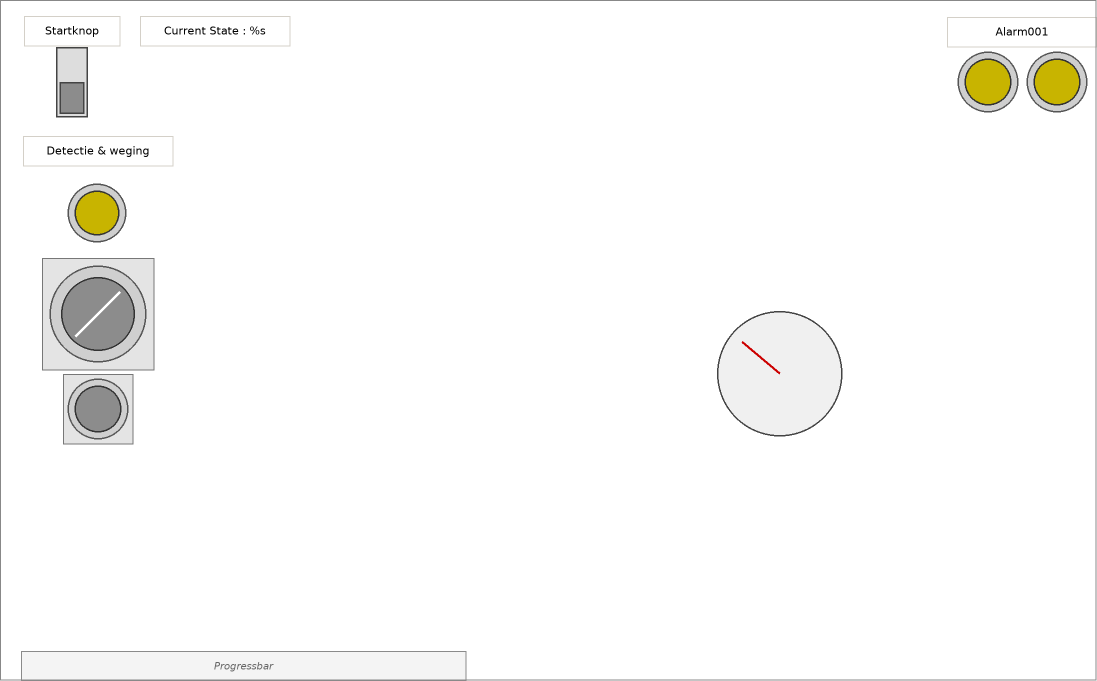
VISUALIZATION Overview  // 1097x681
    Meter180 (657,311 245x125), value: GVL.geschrevenSnelheid, style: Meter-Meter180-Gray, scale format: %.1f, scale 0..200
    Progressbar (21,651 445x30)
    Potentiometer360 (42,254 112x120), variable: GVL.weegcelWaarde, style: Potentiometer-Potentiometer360-Gray, scale format: %.1f, scale 0..100
        p2431819421: Outside
    PushSwitchLed (63,374 70x70), variable: GVL.LS_001, behaviour: TOGGLE, style: Switch-PushSwitchLed-Gray
    Lamp1 (63,178 68x70), variable: GVL.objectDetected, style: Lamp-Lamp1-Yellow
    Textfield (23,136 150x30), "Detectie & weging"
    Group (24,16 96x101)
        Textfield (0,0 96x30), "Startknop", text variable: MAIN.Modus
        DipSwitch (13,31 70x70), variable: GVL.KN_001, behaviour: TOGGLE, style: Switch-DipSwitch-Gray
    Group (947,17 150x100)
        Group (6,30 139x70)
            Lamp1 (0,0 70x70), variable: GVL.ALM001, style: Lamp-Lamp1-Yellow
            Lamp1 (69,0 70x70), variable: GVL.alarmActief, style: Lamp-Lamp1-Yellow
        Textfield (0,0 150x30), "Alarm001"
    Textfield (140,16 150x30), "Current State : %s", text variable: MAIN.Modus
END_VISUALIZATION

(* stored: Version 1.1.0.1, ProductVersion 3.1.4024.12
   Visu Overview: Id {a0e15c2f-f645-4d33-8618-7bbc2738044e} *)
